// TIA Portal V16 export
// export: Created 2023-03-29T11:03:46.9367891Z, ExportSetting WithDefaults, DisplayName Totally Integrated Automation Portal, DisplayVersion V16 Update 6, DisplayName TIA Portal Version Control Interface, DisplayVersion V16 Update 2, DisplayName TIA Portal Openness, DisplayVersion V16 Update 6, DisplayName STEP 7 Professional, DisplayVersion V16 Update 6, DisplayName STEP 7 Safety, DisplayVersion V16, DisplayName WinCC Advanced, DisplayVersion V16 Update 6
VAR_GLOBAL   // PLC tag table "ModbusTCP"
   memTrig_Client_ReceivingTIME AT %M206.4 : Bool;
   memTrig_Step_Sending AT %M9.4 : Bool;   // Pamieć zbocza na uruchomienie pętli Modbus TCP wysyłanie
   done_modbusTCP_przetworzone AT %M9.1 : Bool;   // bit zezwala na wysłanie danych po przetworzeniu przez program PLC Zasuwy
   memTrig_Step_Receiving_Time AT %M9.6 : Bool;   // Pamieć zbocza na uruchomienie pętli Modbus TCP pobieranie Time
   memTrig_Step_Receiving AT %M9.5 : Bool;   // Pamieć zbocza na uruchomienie pętli Modbus TCP pobieranie
   memRisingTriger_Data_13 AT %M208.4 : Bool;   // pamieć zbocza zmiany danych w zmiennej
   memRisingTriger_Data_9 AT %M208.0 : Bool;   // pamieć zbocza zmiany danych w zmiennej
   memRisingTriger_Data_6 AT %M207.5 : Bool;   // pamieć zbocza zmiany danych w zmiennej
   memRisingTriger_Data_5 AT %M207.4 : Bool;   // pamieć zbocza zmiany danych w zmiennej
   memRisingTriger_Data_7 AT %M207.6 : Bool;   // pamieć zbocza zmiany danych w zmiennej
   memRisingTriger_Data_10 AT %M208.1 : Bool;   // pamieć zbocza zmiany danych w zmiennej
   memRisingTriger_Data_8 AT %M207.7 : Bool;   // pamieć zbocza zmiany danych w zmiennej
   memRisingTriger_Data_11 AT %M208.2 : Bool;   // pamieć zbocza zmiany danych w zmiennej
   memRisingTriger_Data_1 AT %M207.0 : Bool;   // pamieć zbocza zmiany danych w zmiennej
   memRisingTriger_Data_2 AT %M207.1 : Bool;   // pamieć zbocza zmiany danych w zmiennej
   memRisingTriger_Data_4 AT %M207.3 : Bool;   // pamieć zbocza zmiany danych w zmiennej
   memRisingTriger_Data_12 AT %M208.3 : Bool;   // pamieć zbocza zmiany danych w zmiennej
   memRisingTriger_Data_3 AT %M207.2 : Bool;   // pamieć zbocza zmiany danych w zmiennej
   memRisingTriger_Data_1_2 AT %M212.4 : Bool;   // pamieć zbocza zmiany danych w zmiennej
   memTrig_SendingError_4 AT %M210.7 : Bool;   // bit pamęci zbocza błedu wysyłania modbus tCP
   memTrig_Client_Receiving_12 AT %M210.1 : Bool;   // pamieć zbocza zmiany danych w zmiennej
   memTrig_Client_Receiving_3 AT %M209.0 : Bool;   // pamieć zbocza zmiany danych w zmiennej
   memTrig_Client_Receiving_9 AT %M209.6 : Bool;   // pamieć zbocza zmiany danych w zmiennej
   memTrig_Client_Receiving_11 AT %M210.0 : Bool;   // pamieć zbocza zmiany danych w zmiennej
   memTrig_Step_Sending_1 AT %M211.0 : Bool;   // Pamieć zbocza na uruchomienie pętli Modbus TCP wysyłanie
   memTrig_Client_Receiving_6 AT %M209.3 : Bool;   // pamieć zbocza zmiany danych w zmiennej
   memTrig_Client_Receiving_4 AT %M209.1 : Bool;   // pamieć zbocza zmiany danych w zmiennej
   done_modbusTCP_przetw_1 AT %M211.1 : Bool;   // bit zezwala na wysłanie danych po przetworzeniu przez program PLC Zasuwy
   memTrig_SendingError_2 AT %M210.5 : Bool;   // bit pamęci zbocza błedu wysyłania modbus tCP
   done_modbusTCP_przetw_6 AT %M212.2 : Bool;   // bit zezwala na wysłanie danych po przetworzeniu przez program PLC Zasuwy
   memTrig_Client_Receiving_2 AT %M208.7 : Bool;   // pamieć zbocza zmiany danych w zmiennej
   done_modbusTCP_przetw_4 AT %M212.0 : Bool;   // bit zezwala na wysłanie danych po przetworzeniu przez program PLC Zasuwy
   done_modbusTCP_przetw_2 AT %M211.2 : Bool;   // bit zezwala na wysłanie danych po przetworzeniu przez program PLC Zasuwy
   memTrig_Client_Receiving_7 AT %M209.4 : Bool;   // pamieć zbocza zmiany danych w zmiennej
   memTrig_Client_Receiving_13 AT %M210.2 : Bool;   // pamieć zbocza zmiany danych w zmiennej
   memRisingTriger_Data_1_1 AT %M212.3 : Bool;   // pamieć zbocza zmiany danych w zmiennej
   memTrig_Client_Receiving_5 AT %M209.2 : Bool;   // pamieć zbocza zmiany danych w zmiennej
   memRisingTriger_Data_1_5 AT %M212.7 : Bool;   // pamieć zbocza zmiany danych w zmiennej
   memTrig_Client_Receiving_1 AT %M208.6 : Bool;   // pamieć zbocza zmiany danych w zmiennej
   memTrig_Step_Sending_4 AT %M211.6 : Bool;   // Pamieć zbocza na uruchomienie pętli Modbus TCP wysyłanie
   memTrig_Client_Receiving_10 AT %M209.7 : Bool;   // pamieć zbocza zmiany danych w zmiennej
   memRisingTriger_Data_1_4 AT %M212.6 : Bool;   // pamieć zbocza zmiany danych w zmiennej
   memTrig_Client_Receiving_8 AT %M209.5 : Bool;   // pamieć zbocza zmiany danych w zmiennej
   memTrig_SendingError_3 AT %M210.6 : Bool;   // bit pamęci zbocza błedu wysyłania modbus tCP
   memTrig_Step_Sending_5 AT %M211.7 : Bool;   // Pamieć zbocza na uruchomienie pętli Modbus TCP wysyłanie
   done_modbusTCP_przetw_3 AT %M211.3 : Bool;   // bit zezwala na wysłanie danych po przetworzeniu przez program PLC Zasuwy
   memRisingTriger_Data_1_3 AT %M212.5 : Bool;   // pamieć zbocza zmiany danych w zmiennej
   memTrig_Step_Sending_2 AT %M211.4 : Bool;   // Pamieć zbocza na uruchomienie pętli Modbus TCP wysyłanie
   done_modbusTCP_przetw_5 AT %M212.1 : Bool;   // bit zezwala na wysłanie danych po przetworzeniu przez program PLC Zasuwy
   memTrig_SendingError_1 AT %M210.4 : Bool;   // bit pamęci zbocza błedu wysyłania modbus tCP
   memTrig_Client_Receiving_14 AT %M210.3 : Bool;   // pamieć zbocza zmiany danych w zmiennej
   memTrig_Step_Sending_3 AT %M211.5 : Bool;   // Pamieć zbocza na uruchomienie pętli Modbus TCP wysyłanie
   memTrig_Error_Receiving AT %M208.5 : Bool;   // pamieć zboczawystąpienia błędu pobierania
   memRisingTriger_Data_16 AT %M213.2 : Bool;   // pamieć zbocza zmiany danych w zmiennej
   memTrig_Client_Receiving_15 AT %M213.3 : Bool;   // pamieć zbocza zmiany danych w zmiennej
   memRisingTriger_Data_14 AT %M213.0 : Bool;   // pamieć zbocza zmiany danych w zmiennej
   memTrig_Client_Receiving_16 AT %M213.4 : Bool;   // pamieć zbocza zmiany danych w zmiennej
   memRisingTriger_Data_15 AT %M213.1 : Bool;   // pamieć zbocza zmiany danych w zmiennej
   memTrig_loop_error AT %M206.5 : Bool;   // błąd petli Modbus TCP brak obiegu pętli
   memRisingTriger_Data_50 AT %M227.1 : Bool;
   memTrig_Client_Receiving_37 AT %M216.4 : Bool;   // pamieć zbocza zmiany danych w zmiennej
   memRisingTriger_Data_83 AT %M231.2 : Bool;
   memTrig_Client_Receiving_84 AT %M222.3 : Bool;   // pamieć zbocza zmiany danych w zmiennej
   memRisingTriger_Data_76 AT %M230.3 : Bool;
   memRisingTriger_Data_18 AT %M223.1 : Bool;
   memTrig_Client_Receiving_38 AT %M216.5 : Bool;   // pamieć zbocza zmiany danych w zmiennej
   memRisingTriger_Data_89 AT %M232.0 : Bool;
   memTrig_Client_Receiving_17 AT %M214.0 : Bool;   // pamieć zbocza zmiany danych w zmiennej
   memTrig_Client_Receiving_81 AT %M222.0 : Bool;   // pamieć zbocza zmiany danych w zmiennej
   memRisingTriger_Data_81 AT %M231.0 : Bool;
   memTrig_Client_Receiving_66 AT %M220.1 : Bool;   // pamieć zbocza zmiany danych w zmiennej
   memTrig_Client_Receiving_62 AT %M219.5 : Bool;   // pamieć zbocza zmiany danych w zmiennej
   memTrig_Client_Receiving_21 AT %M214.4 : Bool;   // pamieć zbocza zmiany danych w zmiennej
   memTrig_Client_Receiving_65 AT %M220.0 : Bool;   // pamieć zbocza zmiany danych w zmiennej
   memTrig_Client_Receiving_43 AT %M217.2 : Bool;   // pamieć zbocza zmiany danych w zmiennej
   memRisingTriger_Data_85 AT %M231.4 : Bool;
   memTrig_Client_Receiving_25 AT %M215.0 : Bool;   // pamieć zbocza zmiany danych w zmiennej
   memRisingTriger_Data_70 AT %M229.5 : Bool;
   memTrig_Client_Receiving_46 AT %M217.5 : Bool;   // pamieć zbocza zmiany danych w zmiennej
   memTrig_Client_Receiving_47 AT %M217.6 : Bool;   // pamieć zbocza zmiany danych w zmiennej
   memTrig_Client_Receiving_18 AT %M214.1 : Bool;   // pamieć zbocza zmiany danych w zmiennej
   memRisingTriger_Data_40 AT %M225.7 : Bool;
   memRisingTriger_Data_86 AT %M231.5 : Bool;
   memRisingTriger_Data_68 AT %M229.3 : Bool;
   memTrig_Client_Receiving_19 AT %M214.2 : Bool;   // pamieć zbocza zmiany danych w zmiennej
   memTrig_Client_Receiving_41 AT %M217.0 : Bool;   // pamieć zbocza zmiany danych w zmiennej
   memRisingTriger_Data_45 AT %M226.4 : Bool;
   memTrig_Client_Receiving_64 AT %M219.7 : Bool;   // pamieć zbocza zmiany danych w zmiennej
   memRisingTriger_Data_28 AT %M224.3 : Bool;
   memTrig_Client_Receiving_49 AT %M218.0 : Bool;   // pamieć zbocza zmiany danych w zmiennej
   memRisingTriger_Data_65 AT %M229.0 : Bool;
   memTrig_Client_Receiving_35 AT %M216.2 : Bool;   // pamieć zbocza zmiany danych w zmiennej
   memRisingTriger_Data_21 AT %M223.4 : Bool;
   memTrig_Client_Receiving_72 AT %M220.7 : Bool;   // pamieć zbocza zmiany danych w zmiennej
   memTrig_Client_Receiving_57 AT %M219.0 : Bool;   // pamieć zbocza zmiany danych w zmiennej
   memTrig_Client_Receiving_51 AT %M218.2 : Bool;   // pamieć zbocza zmiany danych w zmiennej
   memTrig_Client_Receiving_28 AT %M215.3 : Bool;   // pamieć zbocza zmiany danych w zmiennej
   memRisingTriger_Data_66 AT %M229.1 : Bool;
   memTrig_Client_Receiving_45 AT %M217.4 : Bool;   // pamieć zbocza zmiany danych w zmiennej
   memTrig_Client_Receiving_89 AT %M223.0 : Bool;   // pamieć zbocza zmiany danych w zmiennej
   memRisingTriger_Data_35 AT %M225.2 : Bool;
   memTrig_Client_Receiving_83 AT %M222.2 : Bool;   // pamieć zbocza zmiany danych w zmiennej
   memRisingTriger_Data_56 AT %M227.7 : Bool;
   memRisingTriger_Data_20 AT %M223.3 : Bool;
   memTrig_Client_Receiving_36 AT %M216.3 : Bool;   // pamieć zbocza zmiany danych w zmiennej
   memTrig_Client_Receiving_26 AT %M215.1 : Bool;   // pamieć zbocza zmiany danych w zmiennej
   memRisingTriger_Data_23 AT %M223.6 : Bool;
   memRisingTriger_Data_48 AT %M226.7 : Bool;
   memRisingTriger_Data_64 AT %M228.7 : Bool;
   memRisingTriger_Data_61 AT %M228.4 : Bool;
   memRisingTriger_Data_36 AT %M225.3 : Bool;
   memRisingTriger_Data_88 AT %M231.7 : Bool;
   memTrig_Client_Receiving_76 AT %M221.3 : Bool;   // pamieć zbocza zmiany danych w zmiennej
   memRisingTriger_Data_72 AT %M229.7 : Bool;
   memRisingTriger_Data_74 AT %M230.1 : Bool;
   memRisingTriger_Data_39 AT %M225.6 : Bool;
   memRisingTriger_Data_90 AT %M232.1 : Bool;
   memRisingTriger_Data_25 AT %M224.0 : Bool;
   memRisingTriger_Data_44 AT %M226.3 : Bool;
   memRisingTriger_Data_80 AT %M230.7 : Bool;
   memTrig_Client_Receiving_70 AT %M220.5 : Bool;   // pamieć zbocza zmiany danych w zmiennej
   memRisingTriger_Data_37 AT %M225.4 : Bool;
   memTrig_Client_Receiving_20 AT %M214.3 : Bool;   // pamieć zbocza zmiany danych w zmiennej
   memTrig_Client_Receiving_34 AT %M216.1 : Bool;   // pamieć zbocza zmiany danych w zmiennej
   memRisingTriger_Data_49 AT %M227.0 : Bool;
   memRisingTriger_Data_78 AT %M230.5 : Bool;
   memRisingTriger_Data_38 AT %M225.5 : Bool;
   memTrig_Client_Receiving_87 AT %M222.6 : Bool;   // pamieć zbocza zmiany danych w zmiennej
   memTrig_Client_Receiving_30 AT %M215.5 : Bool;   // pamieć zbocza zmiany danych w zmiennej
   memRisingTriger_Data_42 AT %M226.1 : Bool;
   memRisingTriger_Data_57 AT %M228.0 : Bool;
   memTrig_Client_Receiving_54 AT %M218.5 : Bool;   // pamieć zbocza zmiany danych w zmiennej
   memRisingTriger_Data_77 AT %M230.4 : Bool;
   memTrig_Client_Receiving_86 AT %M222.5 : Bool;   // pamieć zbocza zmiany danych w zmiennej
   memTrig_Client_Receiving_63 AT %M219.6 : Bool;   // pamieć zbocza zmiany danych w zmiennej
   memTrig_Client_Receiving_67 AT %M220.2 : Bool;   // pamieć zbocza zmiany danych w zmiennej
   memTrig_Client_Receiving_75 AT %M221.2 : Bool;   // pamieć zbocza zmiany danych w zmiennej
   memRisingTriger_Data_54 AT %M227.5 : Bool;
   memTrig_Client_Receiving_24 AT %M214.7 : Bool;   // pamieć zbocza zmiany danych w zmiennej
   memRisingTriger_Data_41 AT %M226.0 : Bool;
   memTrig_Client_Receiving_82 AT %M222.1 : Bool;   // pamieć zbocza zmiany danych w zmiennej
   memRisingTriger_Data_75 AT %M230.2 : Bool;
   memTrig_Client_Receiving_61 AT %M219.4 : Bool;   // pamieć zbocza zmiany danych w zmiennej
   memRisingTriger_Data_59 AT %M228.2 : Bool;
   memRisingTriger_Data_33 AT %M225.0 : Bool;
   memRisingTriger_Data_19 AT %M223.2 : Bool;
   memTrig_Client_Receiving_56 AT %M218.7 : Bool;   // pamieć zbocza zmiany danych w zmiennej
   memTrig_Client_Receiving_88 AT %M222.7 : Bool;   // pamieć zbocza zmiany danych w zmiennej
   memRisingTriger_Data_47 AT %M226.6 : Bool;
   memTrig_Client_Receiving_59 AT %M219.2 : Bool;   // pamieć zbocza zmiany danych w zmiennej
   memTrig_Client_Receiving_48 AT %M217.7 : Bool;   // pamieć zbocza zmiany danych w zmiennej
   memTrig_Client_Receiving_23 AT %M214.6 : Bool;   // pamieć zbocza zmiany danych w zmiennej
   memTrig_Client_Receiving_32 AT %M215.7 : Bool;   // pamieć zbocza zmiany danych w zmiennej
   memTrig_Client_Receiving_53 AT %M218.4 : Bool;   // pamieć zbocza zmiany danych w zmiennej
   memRisingTriger_Data_79 AT %M230.6 : Bool;
   memRisingTriger_Data_43 AT %M226.2 : Bool;
   memRisingTriger_Data_73 AT %M230.0 : Bool;
   memRisingTriger_Data_87 AT %M231.6 : Bool;
   memRisingTriger_Data_58 AT %M228.1 : Bool;
   memRisingTriger_Data_69 AT %M229.4 : Bool;
   memTrig_Client_Receiving_42 AT %M217.1 : Bool;   // pamieć zbocza zmiany danych w zmiennej
   memTrig_Client_Receiving_69 AT %M220.4 : Bool;   // pamieć zbocza zmiany danych w zmiennej
   memTrig_Client_Receiving_44 AT %M217.3 : Bool;   // pamieć zbocza zmiany danych w zmiennej
   memTrig_Client_Receiving_85 AT %M222.4 : Bool;   // pamieć zbocza zmiany danych w zmiennej
   memTrig_Client_Receiving_31 AT %M215.6 : Bool;   // pamieć zbocza zmiany danych w zmiennej
   memTrig_Client_Receiving_27 AT %M215.2 : Bool;   // pamieć zbocza zmiany danych w zmiennej
   memRisingTriger_Data_24 AT %M223.7 : Bool;
   memTrig_Client_Receiving_50 AT %M218.1 : Bool;   // pamieć zbocza zmiany danych w zmiennej
   memRisingTriger_Data_17 AT %M206.6 : Bool;
   memTrig_Client_Receiving_22 AT %M214.5 : Bool;   // pamieć zbocza zmiany danych w zmiennej
   memRisingTriger_Data_52 AT %M227.3 : Bool;
   memRisingTriger_Data_55 AT %M227.6 : Bool;
   memRisingTriger_Data_34 AT %M225.1 : Bool;
   memTrig_Client_Receiving_77 AT %M221.4 : Bool;   // pamieć zbocza zmiany danych w zmiennej
   memRisingTriger_Data_82 AT %M231.1 : Bool;
   memRisingTriger_Data_67 AT %M229.2 : Bool;
   memRisingTriger_Data_26 AT %M224.1 : Bool;
   memTrig_Client_Receiving_60 AT %M219.3 : Bool;   // pamieć zbocza zmiany danych w zmiennej
   memRisingTriger_Data_27 AT %M224.2 : Bool;
   memTrig_Client_Receiving_52 AT %M218.3 : Bool;   // pamieć zbocza zmiany danych w zmiennej
   memRisingTriger_Data_84 AT %M231.3 : Bool;
   memTrig_Client_Receiving_29 AT %M215.4 : Bool;   // pamieć zbocza zmiany danych w zmiennej
   memTrig_Client_Receiving_73 AT %M221.0 : Bool;   // pamieć zbocza zmiany danych w zmiennej
   memRisingTriger_Data_62 AT %M228.5 : Bool;
   memTrig_Client_Receiving_58 AT %M219.1 : Bool;   // pamieć zbocza zmiany danych w zmiennej
   memRisingTriger_Data_71 AT %M229.6 : Bool;
   memTrig_Client_Receiving_79 AT %M221.6 : Bool;   // pamieć zbocza zmiany danych w zmiennej
   memTrig_Client_Receiving_33 AT %M216.0 : Bool;   // pamieć zbocza zmiany danych w zmiennej
   memRisingTriger_Data_22 AT %M223.5 : Bool;
   memTrig_Client_Receiving_74 AT %M221.1 : Bool;   // pamieć zbocza zmiany danych w zmiennej
   memRisingTriger_Data_51 AT %M227.2 : Bool;
   memTrig_Client_Receiving_78 AT %M221.5 : Bool;   // pamieć zbocza zmiany danych w zmiennej
   memTrig_Client_Receiving_55 AT %M218.6 : Bool;   // pamieć zbocza zmiany danych w zmiennej
   memRisingTriger_Data_30 AT %M224.5 : Bool;
   memTrig_Client_Receiving_40 AT %M216.7 : Bool;   // pamieć zbocza zmiany danych w zmiennej
   memRisingTriger_Data_53 AT %M227.4 : Bool;
   memRisingTriger_Data_29 AT %M224.4 : Bool;
   memRisingTriger_Data_32 AT %M224.7 : Bool;
   memRisingTriger_Data_46 AT %M226.5 : Bool;
   memRisingTriger_Data_60 AT %M228.3 : Bool;
   memRisingTriger_tmerDisconected AT %M228.6 : Bool;   // znacznik załączenia opóźnienia
   timerDISCONECTED_TCP_SERVER_1 AT %M216.6 : Bool;   // znacznik opoźnienia rozłączenia tcp modbus
   timerDISCONECTED_TCP_SERVER_2 AT %M220.3 : Bool;   // znacznik opoźnienia rozłączenia tcp modbus
   timerDISCONECTED_TCP_SERVER_3 AT %M220.6 : Bool;   // znacznik opoźnienia rozłączenia tcp modbus
   timerDISCONECTED_TCP_SERVER_4 AT %M221.7 : Bool;   // znacznik opoźnienia rozłączenia tcp modbus
   memRisingTriger_resetModbusTCP AT %M224.6 : Bool;   // znacznik przerwania połaczenia Modbus TCP na 10sek
END_VAR
